// TIA Portal V18 export
DATA_BLOCK "HSsAI"   // DB1021
{ S7_Optimized_Access := 'FALSE' }
VERSION : 0.1
// stored: AutoNumber false, DBAccessibleFromOPCUA true, IsOnlyStoredInLoadMemory false, IsWriteProtectedInAS false
   VAR
      AI : "UDT_HSsAI";
   END_VAR
BEGIN
END_DATA_BLOCK
